// TIA Portal V17 export
// export: Created 2024-09-15T12:30:35.3253192Z, ExportSetting WithDefaults, DisplayName Totally Integrated Automation Portal, DisplayVersion V17, DisplayName TIA Portal Openness, DisplayVersion V17, DisplayName TIA Portal Version Control Interface, DisplayVersion V17, DisplayName STEP 7 Professional, DisplayVersion V17, DisplayName STEP 7 Safety, DisplayVersion V17, DisplayName WinCC Professional, DisplayVersion V17
TYPE "typ_Workpiece_States"
// stored: IsFailsafeCompliant false
   STRUCT
      x_inOven : Bool;   // Workpiece is int the oven
      ldt_Oven : LDT;   // Timestamp for workpiece going in/out oven
      x_ColorObserved : Bool;   // A new color has been observed
      s_ObservedColor : String;   // Color observed at color sensor ("RED"/"WHITE"/"BLUE")
      w_ObservedColorValue : Word;   // Value of color sensor
      ldt_Color : LDT;   // Timestamp of color observation
      x_atSaw : Bool;   // Workpiece is at the saw
      ldt_Saw : LDT;   // Timestamp for workpiece arriving at/ leaving saw
      x_onTransportBelt : Bool;   // Workpiece is on the sorting line
      ldt_TransportBelt : LDT;   // Timestamp for workpiece going on/off sorting line
   END_STRUCT;
END_TYPE
